// TIA Portal V16 export
// export: Created 2023-05-08T20:00:19.0935246Z, ExportSetting WithDefaults, DisplayName Totally Integrated Automation Portal, DisplayVersion V16 Update 6, DisplayName TIA Portal Version Control Interface, DisplayVersion V16 Update 2, DisplayName TIA Portal Openness, DisplayVersion V16 Update 6, DisplayName STEP 7 Professional, DisplayVersion V16 Update 6, DisplayName STEP 7 Safety, DisplayVersion V16, DisplayName WinCC Advanced, DisplayVersion V16 Update 6
VAR_GLOBAL   // PLC tag table "HVOEin_Aus"
   S1 AT %I0.1 : Bool;   // Schalter Aus Ein
   S5 AT %I0.2 : Bool;   // Start Quittieren NO
   S2 AT %I0.3 : Bool;   // Automatik NO
   S3 AT %I0.4 : Bool;   // Hand NO
   S4 AT %I0.5 : Bool;   // Stopp NC
   P5 AT %Q0.0 : Bool;   // Betrieb Meldeleuchte
   P2 AT %Q0.1 : Bool;   // St�rung Meldeleuchte
   P1 AT %Q0.2 : Bool;   // Automatik Meldeleuchte
   P3 AT %Q0.3 : Bool;   // Hand Meldeleuchte
   P4 AT %Q0.4 : Bool;   // Stopp Meldeleuchte
   S0 AT %I0.0 : Bool;   // Not Aus
   SollPos AT %IW256 : Int;   // Soll Position INT gewandelt
   IstPos AT %QW256 : Int;   // Ist Position INT
   Betriebsarten AT %IW258 : Int;
END_VAR
